// TIA Portal V17 export
// export: Created 2025-03-10T12:16:33.0692349Z, ExportSetting WithDefaults, DisplayName Totally Integrated Automation Portal, DisplayVersion V17 Update 8, DisplayName TIA Portal Openness, DisplayVersion V17 Update 8, DisplayName TIA Portal Version Control Interface, DisplayVersion V17, DisplayName SINAMICS Startdrive Advanced, DisplayVersion V17 SP2, DisplayName SINAMICS Startdrive G110M, G120, G120C, G120D, G120P, G115D, DisplayVersion V17 SP2, DisplayName SINAMICS Startdrive G130, G150, S120, S150, SINAMICS MV, S210, DisplayVersion V17 SP2, DisplayName STEP 7 Professional, DisplayVersion V17 Update 8, DisplayName SINUMERIK ONE STEP 7 Toolbox, DisplayVersion V17 Update 12, DisplayName SINUMERIK 840D sl STEP 7 Toolbox, DisplayVersion V17 Update 12, DisplayName STEP 7 Safety, DisplayVersion V17 Update 6, DisplayName WinCC Advanced, DisplayVersion V17 Update 8
FUNCTION "FC1453_LASER_COOLING_SYSTEM" : Void   // FC1453, LAD
{ S7_Optimized_Access := 'FALSE' }
VERSION : 0.1
// stored: AutoNumber false, IsIECCheckEnabled false, SetENOAutomatically false, UDAEnableTagReadback false
   VAR_TEMP
      COOLING_FLOW_AUX : Real;
      COOLING_FLOW_AUX_1 : Real;
      COOLING_FLOW_AUX_2 : Int;
      COOLING_TEMP_AUX : Real;
      COOLING_TEMP_AUX_1 : Real;
   END_VAR
BEGIN

REGION Network 1: CALL FB1453 LASER COOLING UNIT 01
   // 2#0000_0001 OPTIONS 0 BIT 0 LASER OUTPUT FLOW LOW ALARM GIVEN BY BIT INPUT
   // 2#0000_0010 OPTIONS 0 BIT 1 NOZZLE FLOW LOW ALARM GIVEN BY BIT INPUT
   // 2#0000_0100 OPTIONS 0 BIT 2 HEAD FLOW LOW ALARM GIVEN BY BIT INPUT
   // 2#0000_1000 OPTIONS 0 BIT 3 LASER OUTPUT FLOW ALARMS GIVEN BY ANALOG VALUE
   // 2#0001_0000 OPTIONS 0 BIT 4 NOZZLE FLOW ALARMS GIVEN BY ANALOG VALUE
   // 2#0010_0000 OPTIONS 0 BIT 5 HEAD FLOW ALARMS GIVEN BY ANALOG VALUE
   // 2#0100_0000 OPTIONS 0 BIT 6 SPARE
   // 2#1000_0000 OPTIONS 0 BIT 7 SPARE
   // 
   // 2#0000_0001 OPTIONS 1 BIT 0 LASER OUTPUT TEMP HIGH ALARM GIVEN BY BIT INPUT
   // 2#0000_0010 OPTIONS 1 BIT 1 NOOZLE TEMP HIGH ALARM GIVEN BY BIT INPUT
   // 2#0000_0100 OPTIONS 1 BIT 2 HEAD TEMP HIGH ALARM GIVEN BY BIT INPUT
   // 2#0000_1000 OPTIONS 1 BIT 3 LASER OUTPUT TEMP ALARMS GIVEN BY ANALOG VALUE
   // 2#0001_0000 OPTIONS 1 BIT 4 NOZZLE TEMP ALARMS GIVEN BY ANALOG VALUE
   // 2#0010_0000 OPTIONS 1 BIT 5 HEAD TEMP ALARMS GIVEN BY ANALOG VALUE
   // 2#0100_0000 OPTIONS 1 BIT 6 SPARE OPTION
   // 2#1000_0000 OPTIONS 1 BIT 7 SPARE OPTION
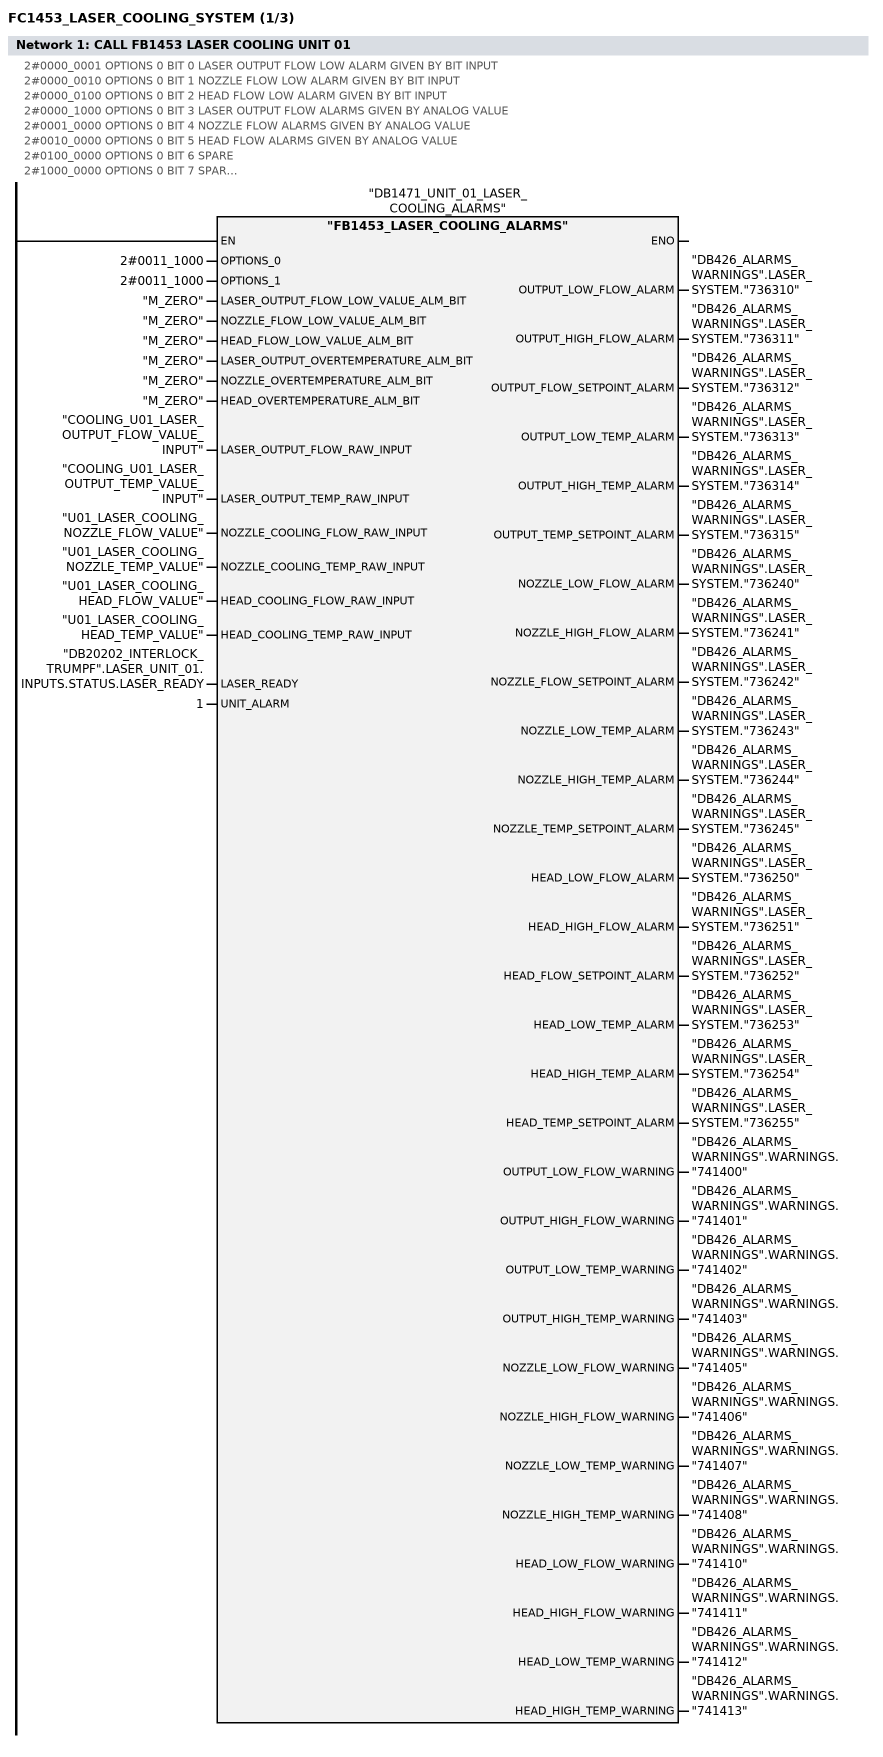
   RUNG wire#powerrail
      "DB1471_UNIT_01_LASER_COOLING_ALARMS"(OPTIONS_0 := 2#0011_1000, OPTIONS_1 := 2#0011_1000, LASER_OUTPUT_FLOW_LOW_VALUE_ALM_BIT := "M_ZERO", NOZZLE_FLOW_LOW_VALUE_ALM_BIT := "M_ZERO", HEAD_FLOW_LOW_VALUE_ALM_BIT := "M_ZERO", LASER_OUTPUT_OVERTEMPERATURE_ALM_BIT := "M_ZERO", NOZZLE_OVERTEMPERATURE_ALM_BIT := "M_ZERO", HEAD_OVERTEMPERATURE_ALM_BIT := "M_ZERO", LASER_OUTPUT_FLOW_RAW_INPUT := "COOLING_U01_LASER_OUTPUT_FLOW_VALUE_INPUT", LASER_OUTPUT_TEMP_RAW_INPUT := "COOLING_U01_LASER_OUTPUT_TEMP_VALUE_INPUT", NOZZLE_COOLING_FLOW_RAW_INPUT := "U01_LASER_COOLING_NOZZLE_FLOW_VALUE", NOZZLE_COOLING_TEMP_RAW_INPUT := "U01_LASER_COOLING_NOZZLE_TEMP_VALUE", HEAD_COOLING_FLOW_RAW_INPUT := "U01_LASER_COOLING_HEAD_FLOW_VALUE", HEAD_COOLING_TEMP_RAW_INPUT := "U01_LASER_COOLING_HEAD_TEMP_VALUE", LASER_READY := "DB20202_INTERLOCK_TRUMPF".LASER_UNIT_01.INPUTS.STATUS.LASER_READY, UNIT_ALARM := 1, OUTPUT_LOW_FLOW_ALARM => "DB426_ALARMS_WARNINGS".LASER_SYSTEM."736310", OUTPUT_HIGH_FLOW_ALARM => "DB426_ALARMS_WARNINGS".LASER_SYSTEM."736311", OUTPUT_FLOW_SETPOINT_ALARM => "DB426_ALARMS_WARNINGS".LASER_SYSTEM."736312", OUTPUT_LOW_TEMP_ALARM => "DB426_ALARMS_WARNINGS".LASER_SYSTEM."736313", OUTPUT_HIGH_TEMP_ALARM => "DB426_ALARMS_WARNINGS".LASER_SYSTEM."736314", OUTPUT_TEMP_SETPOINT_ALARM => "DB426_ALARMS_WARNINGS".LASER_SYSTEM."736315", NOZZLE_LOW_FLOW_ALARM => "DB426_ALARMS_WARNINGS".LASER_SYSTEM."736240", NOZZLE_HIGH_FLOW_ALARM => "DB426_ALARMS_WARNINGS".LASER_SYSTEM."736241", NOZZLE_FLOW_SETPOINT_ALARM => "DB426_ALARMS_WARNINGS".LASER_SYSTEM."736242", NOZZLE_LOW_TEMP_ALARM => "DB426_ALARMS_WARNINGS".LASER_SYSTEM."736243", NOZZLE_HIGH_TEMP_ALARM => "DB426_ALARMS_WARNINGS".LASER_SYSTEM."736244", NOZZLE_TEMP_SETPOINT_ALARM => "DB426_ALARMS_WARNINGS".LASER_SYSTEM."736245", HEAD_LOW_FLOW_ALARM => "DB426_ALARMS_WARNINGS".LASER_SYSTEM."736250", HEAD_HIGH_FLOW_ALARM => "DB426_ALARMS_WARNINGS".LASER_SYSTEM."736251", HEAD_FLOW_SETPOINT_ALARM => "DB426_ALARMS_WARNINGS".LASER_SYSTEM."736252", HEAD_LOW_TEMP_ALARM => "DB426_ALARMS_WARNINGS".LASER_SYSTEM."736253", HEAD_HIGH_TEMP_ALARM => "DB426_ALARMS_WARNINGS".LASER_SYSTEM."736254", HEAD_TEMP_SETPOINT_ALARM => "DB426_ALARMS_WARNINGS".LASER_SYSTEM."736255", OUTPUT_LOW_FLOW_WARNING => "DB426_ALARMS_WARNINGS".WARNINGS."741400", OUTPUT_HIGH_FLOW_WARNING => "DB426_ALARMS_WARNINGS".WARNINGS."741401", OUTPUT_LOW_TEMP_WARNING => "DB426_ALARMS_WARNINGS".WARNINGS."741402", OUTPUT_HIGH_TEMP_WARNING => "DB426_ALARMS_WARNINGS".WARNINGS."741403", NOZZLE_LOW_FLOW_WARNING => "DB426_ALARMS_WARNINGS".WARNINGS."741405", NOZZLE_HIGH_FLOW_WARNING => "DB426_ALARMS_WARNINGS".WARNINGS."741406", NOZZLE_LOW_TEMP_WARNING => "DB426_ALARMS_WARNINGS".WARNINGS."741407", NOZZLE_HIGH_TEMP_WARNING => "DB426_ALARMS_WARNINGS".WARNINGS."741408", HEAD_LOW_FLOW_WARNING => "DB426_ALARMS_WARNINGS".WARNINGS."741410", HEAD_HIGH_FLOW_WARNING => "DB426_ALARMS_WARNINGS".WARNINGS."741411", HEAD_LOW_TEMP_WARNING => "DB426_ALARMS_WARNINGS".WARNINGS."741412", HEAD_HIGH_TEMP_WARNING => "DB426_ALARMS_WARNINGS".WARNINGS."741413")
   END_RUNG
   // the same network as SCL:
   "DB1471_UNIT_01_LASER_COOLING_ALARMS"(OPTIONS_0 := 2#0011_1000,   // "FB1453_LASER_COOLING_ALARMS"
                           OPTIONS_1 := 2#0011_1000,
                           LASER_OUTPUT_FLOW_LOW_VALUE_ALM_BIT := "M_ZERO",
                           NOZZLE_FLOW_LOW_VALUE_ALM_BIT := "M_ZERO",
                           HEAD_FLOW_LOW_VALUE_ALM_BIT := "M_ZERO",
                           LASER_OUTPUT_OVERTEMPERATURE_ALM_BIT := "M_ZERO",
                           NOZZLE_OVERTEMPERATURE_ALM_BIT := "M_ZERO",
                           HEAD_OVERTEMPERATURE_ALM_BIT := "M_ZERO",
                           LASER_OUTPUT_FLOW_RAW_INPUT := "COOLING_U01_LASER_OUTPUT_FLOW_VALUE_INPUT",
                           LASER_OUTPUT_TEMP_RAW_INPUT := "COOLING_U01_LASER_OUTPUT_TEMP_VALUE_INPUT",
                           NOZZLE_COOLING_FLOW_RAW_INPUT := "U01_LASER_COOLING_NOZZLE_FLOW_VALUE",
                           NOZZLE_COOLING_TEMP_RAW_INPUT := "U01_LASER_COOLING_NOZZLE_TEMP_VALUE",
                           HEAD_COOLING_FLOW_RAW_INPUT := "U01_LASER_COOLING_HEAD_FLOW_VALUE",
                           HEAD_COOLING_TEMP_RAW_INPUT := "U01_LASER_COOLING_HEAD_TEMP_VALUE",
                           LASER_READY := "DB20202_INTERLOCK_TRUMPF".LASER_UNIT_01.INPUTS.STATUS.LASER_READY,
                           UNIT_ALARM := 1,
                           OUTPUT_LOW_FLOW_ALARM => "DB426_ALARMS_WARNINGS".LASER_SYSTEM."736310",
                           OUTPUT_HIGH_FLOW_ALARM => "DB426_ALARMS_WARNINGS".LASER_SYSTEM."736311",
                           OUTPUT_FLOW_SETPOINT_ALARM => "DB426_ALARMS_WARNINGS".LASER_SYSTEM."736312",
                           OUTPUT_LOW_TEMP_ALARM => "DB426_ALARMS_WARNINGS".LASER_SYSTEM."736313",
                           OUTPUT_HIGH_TEMP_ALARM => "DB426_ALARMS_WARNINGS".LASER_SYSTEM."736314",
                           OUTPUT_TEMP_SETPOINT_ALARM => "DB426_ALARMS_WARNINGS".LASER_SYSTEM."736315",
                           NOZZLE_LOW_FLOW_ALARM => "DB426_ALARMS_WARNINGS".LASER_SYSTEM."736240",
                           NOZZLE_HIGH_FLOW_ALARM => "DB426_ALARMS_WARNINGS".LASER_SYSTEM."736241",
                           NOZZLE_FLOW_SETPOINT_ALARM => "DB426_ALARMS_WARNINGS".LASER_SYSTEM."736242",
                           NOZZLE_LOW_TEMP_ALARM => "DB426_ALARMS_WARNINGS".LASER_SYSTEM."736243",
                           NOZZLE_HIGH_TEMP_ALARM => "DB426_ALARMS_WARNINGS".LASER_SYSTEM."736244",
                           NOZZLE_TEMP_SETPOINT_ALARM => "DB426_ALARMS_WARNINGS".LASER_SYSTEM."736245",
                           HEAD_LOW_FLOW_ALARM => "DB426_ALARMS_WARNINGS".LASER_SYSTEM."736250",
                           HEAD_HIGH_FLOW_ALARM => "DB426_ALARMS_WARNINGS".LASER_SYSTEM."736251",
                           HEAD_FLOW_SETPOINT_ALARM => "DB426_ALARMS_WARNINGS".LASER_SYSTEM."736252",
                           HEAD_LOW_TEMP_ALARM => "DB426_ALARMS_WARNINGS".LASER_SYSTEM."736253",
                           HEAD_HIGH_TEMP_ALARM => "DB426_ALARMS_WARNINGS".LASER_SYSTEM."736254",
                           HEAD_TEMP_SETPOINT_ALARM => "DB426_ALARMS_WARNINGS".LASER_SYSTEM."736255",
                           OUTPUT_LOW_FLOW_WARNING => "DB426_ALARMS_WARNINGS".WARNINGS."741400",
                           OUTPUT_HIGH_FLOW_WARNING => "DB426_ALARMS_WARNINGS".WARNINGS."741401",
                           OUTPUT_LOW_TEMP_WARNING => "DB426_ALARMS_WARNINGS".WARNINGS."741402",
                           OUTPUT_HIGH_TEMP_WARNING => "DB426_ALARMS_WARNINGS".WARNINGS."741403",
                           NOZZLE_LOW_FLOW_WARNING => "DB426_ALARMS_WARNINGS".WARNINGS."741405",
                           NOZZLE_HIGH_FLOW_WARNING => "DB426_ALARMS_WARNINGS".WARNINGS."741406",
                           NOZZLE_LOW_TEMP_WARNING => "DB426_ALARMS_WARNINGS".WARNINGS."741407",
                           NOZZLE_HIGH_TEMP_WARNING => "DB426_ALARMS_WARNINGS".WARNINGS."741408",
                           HEAD_LOW_FLOW_WARNING => "DB426_ALARMS_WARNINGS".WARNINGS."741410",
                           HEAD_HIGH_FLOW_WARNING => "DB426_ALARMS_WARNINGS".WARNINGS."741411",
                           HEAD_LOW_TEMP_WARNING => "DB426_ALARMS_WARNINGS".WARNINGS."741412",
                           HEAD_HIGH_TEMP_WARNING => "DB426_ALARMS_WARNINGS".WARNINGS."741413");
END_REGION

REGION Network 2: CALL FB1453 LASER COOLING UNIT 02
   // 2#0000_0001 OPTIONS 0 BIT 0 LASER OUTPUT FLOW LOW ALARM GIVEN BY BIT INPUT
   // 2#0000_0010 OPTIONS 0 BIT 1 NOZZLE FLOW LOW ALARM GIVEN BY BIT INPUT
   // 2#0000_0100 OPTIONS 0 BIT 2 HEAD FLOW LOW ALARM GIVEN BY BIT INPUT
   // 2#0000_1000 OPTIONS 0 BIT 3 LASER OUTPUT FLOW ALARMS GIVEN BY ANALOG VALUE
   // 2#0001_0000 OPTIONS 0 BIT 4 NOZZLE FLOW ALARMS GIVEN BY ANALOG VALUE
   // 2#0010_0000 OPTIONS 0 BIT 5 HEAD FLOW ALARMS GIVEN BY ANALOG VALUE
   // 2#0100_0000 OPTIONS 0 BIT 6 SPARE
   // 2#1000_0000 OPTIONS 0 BIT 7 SPARE
   // 
   // 2#0000_0001 OPTIONS 1 BIT 0 LASER OUTPUT TEMP HIGH ALARM GIVEN BY BIT INPUT
   // 2#0000_0010 OPTIONS 1 BIT 1 NOOZLE TEMP HIGH ALARM GIVEN BY BIT INPUT
   // 2#0000_0100 OPTIONS 1 BIT 2 HEAD TEMP HIGH ALARM GIVEN BY BIT INPUT
   // 2#0000_1000 OPTIONS 1 BIT 3 LASER OUTPUT TEMP ALARMS GIVEN BY ANALOG VALUE
   // 2#0001_0000 OPTIONS 1 BIT 4 NOZZLE TEMP ALARMS GIVEN BY ANALOG VALUE
   // 2#0010_0000 OPTIONS 1 BIT 5 HEAD TEMP ALARMS GIVEN BY ANALOG VALUE
   // 2#0100_0000 OPTIONS 1 BIT 6 SPARE OPTION
   // 2#1000_0000 OPTIONS 1 BIT 7 SPARE OPTION
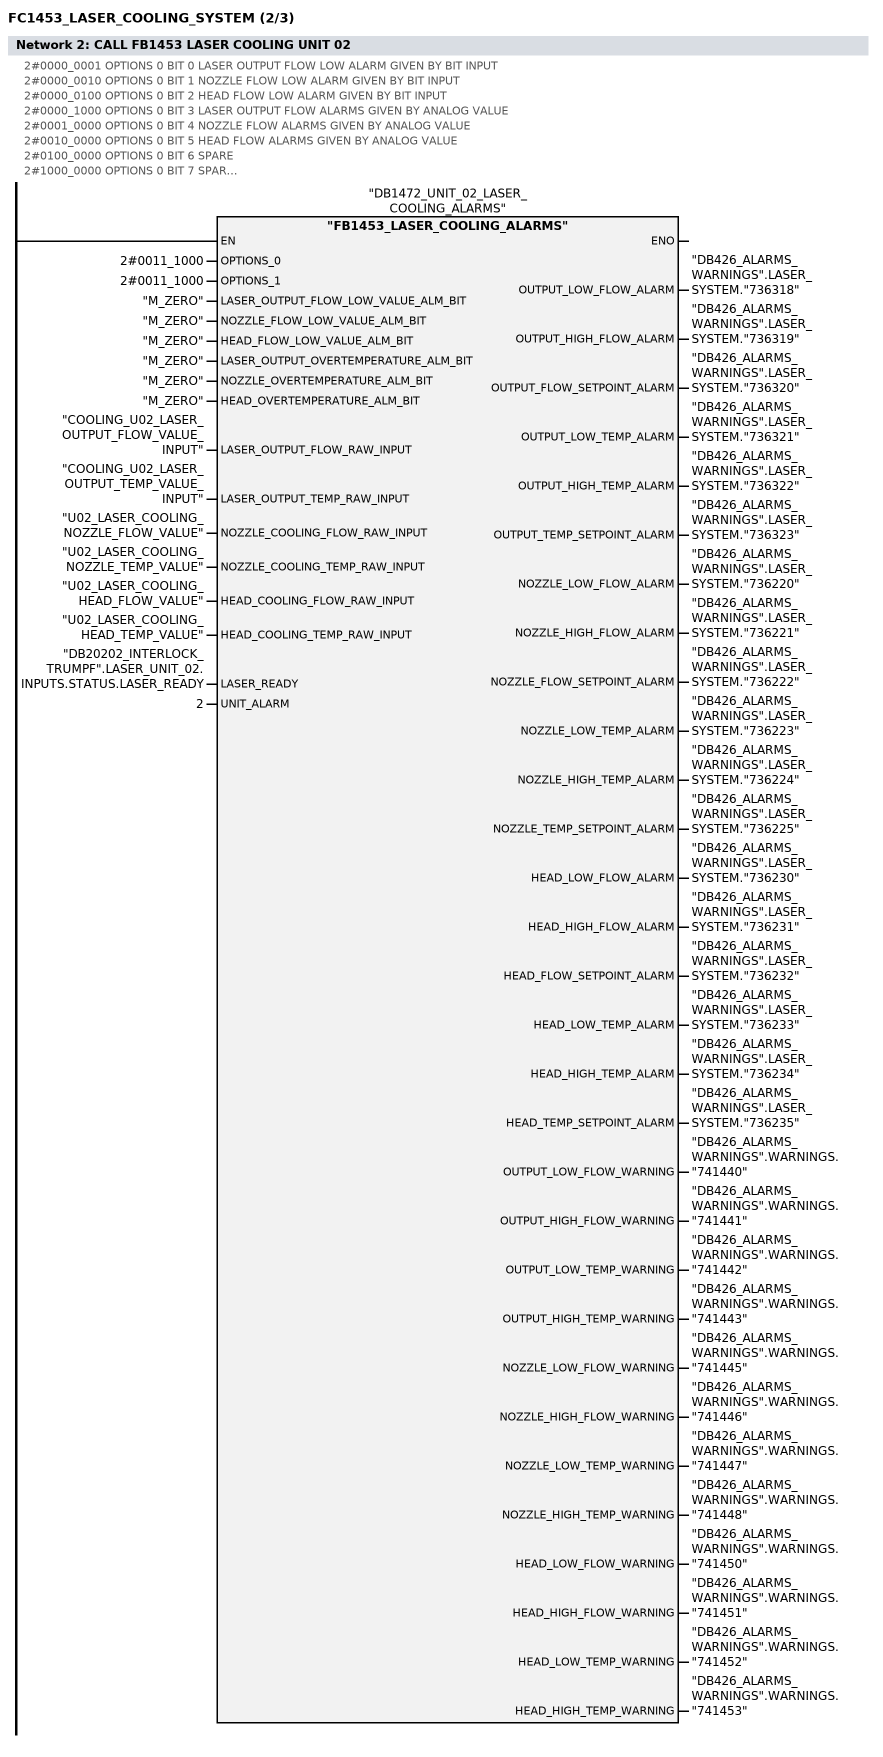
   RUNG wire#powerrail
      "DB1472_UNIT_02_LASER_COOLING_ALARMS"(OPTIONS_0 := 2#0011_1000, OPTIONS_1 := 2#0011_1000, LASER_OUTPUT_FLOW_LOW_VALUE_ALM_BIT := "M_ZERO", NOZZLE_FLOW_LOW_VALUE_ALM_BIT := "M_ZERO", HEAD_FLOW_LOW_VALUE_ALM_BIT := "M_ZERO", LASER_OUTPUT_OVERTEMPERATURE_ALM_BIT := "M_ZERO", NOZZLE_OVERTEMPERATURE_ALM_BIT := "M_ZERO", HEAD_OVERTEMPERATURE_ALM_BIT := "M_ZERO", LASER_OUTPUT_FLOW_RAW_INPUT := "COOLING_U02_LASER_OUTPUT_FLOW_VALUE_INPUT", LASER_OUTPUT_TEMP_RAW_INPUT := "COOLING_U02_LASER_OUTPUT_TEMP_VALUE_INPUT", NOZZLE_COOLING_FLOW_RAW_INPUT := "U02_LASER_COOLING_NOZZLE_FLOW_VALUE", NOZZLE_COOLING_TEMP_RAW_INPUT := "U02_LASER_COOLING_NOZZLE_TEMP_VALUE", HEAD_COOLING_FLOW_RAW_INPUT := "U02_LASER_COOLING_HEAD_FLOW_VALUE", HEAD_COOLING_TEMP_RAW_INPUT := "U02_LASER_COOLING_HEAD_TEMP_VALUE", LASER_READY := "DB20202_INTERLOCK_TRUMPF".LASER_UNIT_02.INPUTS.STATUS.LASER_READY, UNIT_ALARM := 2, OUTPUT_LOW_FLOW_ALARM => "DB426_ALARMS_WARNINGS".LASER_SYSTEM."736318", OUTPUT_HIGH_FLOW_ALARM => "DB426_ALARMS_WARNINGS".LASER_SYSTEM."736319", OUTPUT_FLOW_SETPOINT_ALARM => "DB426_ALARMS_WARNINGS".LASER_SYSTEM."736320", OUTPUT_LOW_TEMP_ALARM => "DB426_ALARMS_WARNINGS".LASER_SYSTEM."736321", OUTPUT_HIGH_TEMP_ALARM => "DB426_ALARMS_WARNINGS".LASER_SYSTEM."736322", OUTPUT_TEMP_SETPOINT_ALARM => "DB426_ALARMS_WARNINGS".LASER_SYSTEM."736323", NOZZLE_LOW_FLOW_ALARM => "DB426_ALARMS_WARNINGS".LASER_SYSTEM."736220", NOZZLE_HIGH_FLOW_ALARM => "DB426_ALARMS_WARNINGS".LASER_SYSTEM."736221", NOZZLE_FLOW_SETPOINT_ALARM => "DB426_ALARMS_WARNINGS".LASER_SYSTEM."736222", NOZZLE_LOW_TEMP_ALARM => "DB426_ALARMS_WARNINGS".LASER_SYSTEM."736223", NOZZLE_HIGH_TEMP_ALARM => "DB426_ALARMS_WARNINGS".LASER_SYSTEM."736224", NOZZLE_TEMP_SETPOINT_ALARM => "DB426_ALARMS_WARNINGS".LASER_SYSTEM."736225", HEAD_LOW_FLOW_ALARM => "DB426_ALARMS_WARNINGS".LASER_SYSTEM."736230", HEAD_HIGH_FLOW_ALARM => "DB426_ALARMS_WARNINGS".LASER_SYSTEM."736231", HEAD_FLOW_SETPOINT_ALARM => "DB426_ALARMS_WARNINGS".LASER_SYSTEM."736232", HEAD_LOW_TEMP_ALARM => "DB426_ALARMS_WARNINGS".LASER_SYSTEM."736233", HEAD_HIGH_TEMP_ALARM => "DB426_ALARMS_WARNINGS".LASER_SYSTEM."736234", HEAD_TEMP_SETPOINT_ALARM => "DB426_ALARMS_WARNINGS".LASER_SYSTEM."736235", OUTPUT_LOW_FLOW_WARNING => "DB426_ALARMS_WARNINGS".WARNINGS."741440", OUTPUT_HIGH_FLOW_WARNING => "DB426_ALARMS_WARNINGS".WARNINGS."741441", OUTPUT_LOW_TEMP_WARNING => "DB426_ALARMS_WARNINGS".WARNINGS."741442", OUTPUT_HIGH_TEMP_WARNING => "DB426_ALARMS_WARNINGS".WARNINGS."741443", NOZZLE_LOW_FLOW_WARNING => "DB426_ALARMS_WARNINGS".WARNINGS."741445", NOZZLE_HIGH_FLOW_WARNING => "DB426_ALARMS_WARNINGS".WARNINGS."741446", NOZZLE_LOW_TEMP_WARNING => "DB426_ALARMS_WARNINGS".WARNINGS."741447", NOZZLE_HIGH_TEMP_WARNING => "DB426_ALARMS_WARNINGS".WARNINGS."741448", HEAD_LOW_FLOW_WARNING => "DB426_ALARMS_WARNINGS".WARNINGS."741450", HEAD_HIGH_FLOW_WARNING => "DB426_ALARMS_WARNINGS".WARNINGS."741451", HEAD_LOW_TEMP_WARNING => "DB426_ALARMS_WARNINGS".WARNINGS."741452", HEAD_HIGH_TEMP_WARNING => "DB426_ALARMS_WARNINGS".WARNINGS."741453")
   END_RUNG
   // the same network as SCL:
   "DB1472_UNIT_02_LASER_COOLING_ALARMS"(OPTIONS_0 := 2#0011_1000,   // "FB1453_LASER_COOLING_ALARMS"
                           OPTIONS_1 := 2#0011_1000,
                           LASER_OUTPUT_FLOW_LOW_VALUE_ALM_BIT := "M_ZERO",
                           NOZZLE_FLOW_LOW_VALUE_ALM_BIT := "M_ZERO",
                           HEAD_FLOW_LOW_VALUE_ALM_BIT := "M_ZERO",
                           LASER_OUTPUT_OVERTEMPERATURE_ALM_BIT := "M_ZERO",
                           NOZZLE_OVERTEMPERATURE_ALM_BIT := "M_ZERO",
                           HEAD_OVERTEMPERATURE_ALM_BIT := "M_ZERO",
                           LASER_OUTPUT_FLOW_RAW_INPUT := "COOLING_U02_LASER_OUTPUT_FLOW_VALUE_INPUT",
                           LASER_OUTPUT_TEMP_RAW_INPUT := "COOLING_U02_LASER_OUTPUT_TEMP_VALUE_INPUT",
                           NOZZLE_COOLING_FLOW_RAW_INPUT := "U02_LASER_COOLING_NOZZLE_FLOW_VALUE",
                           NOZZLE_COOLING_TEMP_RAW_INPUT := "U02_LASER_COOLING_NOZZLE_TEMP_VALUE",
                           HEAD_COOLING_FLOW_RAW_INPUT := "U02_LASER_COOLING_HEAD_FLOW_VALUE",
                           HEAD_COOLING_TEMP_RAW_INPUT := "U02_LASER_COOLING_HEAD_TEMP_VALUE",
                           LASER_READY := "DB20202_INTERLOCK_TRUMPF".LASER_UNIT_02.INPUTS.STATUS.LASER_READY,
                           UNIT_ALARM := 2,
                           OUTPUT_LOW_FLOW_ALARM => "DB426_ALARMS_WARNINGS".LASER_SYSTEM."736318",
                           OUTPUT_HIGH_FLOW_ALARM => "DB426_ALARMS_WARNINGS".LASER_SYSTEM."736319",
                           OUTPUT_FLOW_SETPOINT_ALARM => "DB426_ALARMS_WARNINGS".LASER_SYSTEM."736320",
                           OUTPUT_LOW_TEMP_ALARM => "DB426_ALARMS_WARNINGS".LASER_SYSTEM."736321",
                           OUTPUT_HIGH_TEMP_ALARM => "DB426_ALARMS_WARNINGS".LASER_SYSTEM."736322",
                           OUTPUT_TEMP_SETPOINT_ALARM => "DB426_ALARMS_WARNINGS".LASER_SYSTEM."736323",
                           NOZZLE_LOW_FLOW_ALARM => "DB426_ALARMS_WARNINGS".LASER_SYSTEM."736220",
                           NOZZLE_HIGH_FLOW_ALARM => "DB426_ALARMS_WARNINGS".LASER_SYSTEM."736221",
                           NOZZLE_FLOW_SETPOINT_ALARM => "DB426_ALARMS_WARNINGS".LASER_SYSTEM."736222",
                           NOZZLE_LOW_TEMP_ALARM => "DB426_ALARMS_WARNINGS".LASER_SYSTEM."736223",
                           NOZZLE_HIGH_TEMP_ALARM => "DB426_ALARMS_WARNINGS".LASER_SYSTEM."736224",
                           NOZZLE_TEMP_SETPOINT_ALARM => "DB426_ALARMS_WARNINGS".LASER_SYSTEM."736225",
                           HEAD_LOW_FLOW_ALARM => "DB426_ALARMS_WARNINGS".LASER_SYSTEM."736230",
                           HEAD_HIGH_FLOW_ALARM => "DB426_ALARMS_WARNINGS".LASER_SYSTEM."736231",
                           HEAD_FLOW_SETPOINT_ALARM => "DB426_ALARMS_WARNINGS".LASER_SYSTEM."736232",
                           HEAD_LOW_TEMP_ALARM => "DB426_ALARMS_WARNINGS".LASER_SYSTEM."736233",
                           HEAD_HIGH_TEMP_ALARM => "DB426_ALARMS_WARNINGS".LASER_SYSTEM."736234",
                           HEAD_TEMP_SETPOINT_ALARM => "DB426_ALARMS_WARNINGS".LASER_SYSTEM."736235",
                           OUTPUT_LOW_FLOW_WARNING => "DB426_ALARMS_WARNINGS".WARNINGS."741440",
                           OUTPUT_HIGH_FLOW_WARNING => "DB426_ALARMS_WARNINGS".WARNINGS."741441",
                           OUTPUT_LOW_TEMP_WARNING => "DB426_ALARMS_WARNINGS".WARNINGS."741442",
                           OUTPUT_HIGH_TEMP_WARNING => "DB426_ALARMS_WARNINGS".WARNINGS."741443",
                           NOZZLE_LOW_FLOW_WARNING => "DB426_ALARMS_WARNINGS".WARNINGS."741445",
                           NOZZLE_HIGH_FLOW_WARNING => "DB426_ALARMS_WARNINGS".WARNINGS."741446",
                           NOZZLE_LOW_TEMP_WARNING => "DB426_ALARMS_WARNINGS".WARNINGS."741447",
                           NOZZLE_HIGH_TEMP_WARNING => "DB426_ALARMS_WARNINGS".WARNINGS."741448",
                           HEAD_LOW_FLOW_WARNING => "DB426_ALARMS_WARNINGS".WARNINGS."741450",
                           HEAD_HIGH_FLOW_WARNING => "DB426_ALARMS_WARNINGS".WARNINGS."741451",
                           HEAD_LOW_TEMP_WARNING => "DB426_ALARMS_WARNINGS".WARNINGS."741452",
                           HEAD_HIGH_TEMP_WARNING => "DB426_ALARMS_WARNINGS".WARNINGS."741453");
END_REGION

REGION Network 3: COOLING
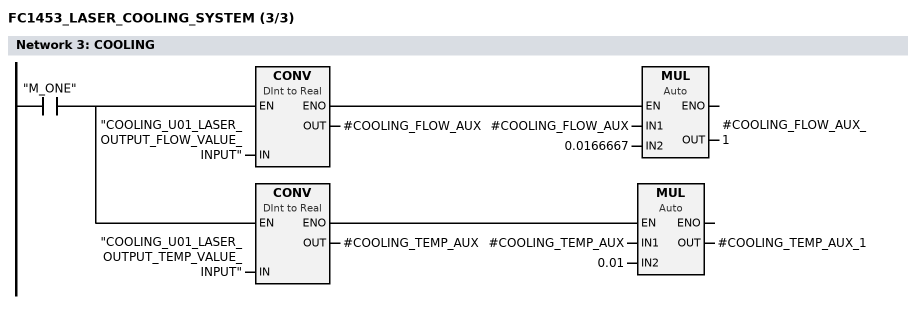
   RUNG wire#powerrail
      Contact( "M_ONE" )
      wire#w1
      { S7_Templates := "[SrcType := DInt, DestType := Real]" } Convert(in := "COOLING_U01_LASER_OUTPUT_FLOW_VALUE_INPUT", out => #COOLING_FLOW_AUX)
      Mul(in1 := #COOLING_FLOW_AUX, in2 := 0.0166667, out => #COOLING_FLOW_AUX_1)
   END_RUNG
   RUNG wire#w1
      { S7_Templates := "[SrcType := DInt, DestType := Real]" } Convert(in := "COOLING_U01_LASER_OUTPUT_TEMP_VALUE_INPUT", out => #COOLING_TEMP_AUX)
      Mul(in1 := #COOLING_TEMP_AUX, in2 := 0.01, out => #COOLING_TEMP_AUX_1)
   END_RUNG
   // the same network as SCL:
   IF "M_ONE" THEN
       #COOLING_FLOW_AUX := DINT_TO_REAL("COOLING_U01_LASER_OUTPUT_FLOW_VALUE_INPUT");
       #COOLING_FLOW_AUX_1 := #COOLING_FLOW_AUX * 0.0166667;
       #COOLING_TEMP_AUX := DINT_TO_REAL("COOLING_U01_LASER_OUTPUT_TEMP_VALUE_INPUT");
       #COOLING_TEMP_AUX_1 := #COOLING_TEMP_AUX * 0.01;
   END_IF;
END_REGION
END_FUNCTION
